// TIA Portal V20 export
DATA_BLOCK "Send_FData_DB"   // DB5
// stored: InstanceOfName Send_FData, InstanceOfType FB
"Send_FData"
   // VAR
   //    TSEND_Instance { S7_SetPoint := 'True'} : TSEND;
   //    status_save { S7_SetPoint := 'True'} : Word;
   //    trigger : Bool;
   // END_VAR
BEGIN
END_DATA_BLOCK
